Fanuc KAREL source: kt00497.KL

-- PROVISIONAL review KL for V1013-1; original PC SHA256 ffd1c98b411f9480be5082ebcf143ee0b176fe3f5449d4d152955ddfab2a76dd
-- Incomplete behavior may be omitted. Consult companion uncertainty JSON. Do not deploy.
PROGRAM KT00497
%NOLOCKGROUP
-- UNRESOLVED_DECL P1 type=000102
-- UNRESOLVED_DECL P2 type=000101
-- UNRESOLVED_DECL OUT type=000199
BEGIN
  -- UNRESOLVED_PC offsets 5-20; opcodes 2E,22,32,35
  -- UNRESOLVED_PC offsets 25-59; opcodes 49,7E,49,60,7E,4A
  -- UNRESOLVED_PC offsets 64-68; opcodes 7F
END KT00497
